FUNCTION_BLOCK FB_GetCPUTemp
VAR_INPUT
	rInterval			: REAL := 10.0;		// [sec]
END_VAR
VAR_OUTPUT
	rCPUTemp			: REAL;				// [deg]
	bError				: BOOL;				// error flag (indicator: error occured)
	nErrID				: UDINT;			// last error ID 
END_VAR
VAR
	// internal use
	sAmsNetId			: STRING := '';		// ADS Net ID (local = '')    
	iState				: INT;
	uData				: UINT;
	stMDP_Addr			: Tc2_MDP.ST_MDP_Addr;
	// FB instances
	fbReadMDPElement	: Tc2_MDP.FB_MDP_ReadElement;  
	tonInterval			: Tc2_Standard.TON;
END_VAR


// Interval timer
tonInterval(IN := NOT tonInterval.Q, PT := REAL_TO_TIME(rInterval * 1000.0));

CASE iState OF
	0: // Initiate program parameters (if required)
		fbReadMDPElement(bExecute := FALSE);
		IF (tonInterval.Q) THEN
			iState := 10;
		END_IF

	10:	// Trigger FB: request CPU data
		stMDP_Addr.nArea := INT_TO_BYTE(Tc2_MDP.eMDP_Area_ConfigArea);
		stMDP_Addr.nTableId := 1;
		stMDP_Addr.nSubIdx := 3;
		fbReadMDPElement(	bExecute := TRUE,
							eModuleType := Tc2_MDP.eMDP_ModT_CPU,
							stMDP_Addr := stMDP_Addr,
							iModIdx := 0,
							pDstBuf := ADR(uData),
							cbDstBufLen := SIZEOF(uData),
							sAmsNetId := sAmsNetId	);
		iState := 20;

	20:	// Process FB: Request CPU temp
		fbReadMDPElement(bExecute := FALSE); 
		IF (NOT fbReadMDPElement.bBusy) THEN
			IF (fbReadMDPElement.bError) THEN
				bError := TRUE;
				nErrID := fbReadMDPElement.nErrID; 
				iState := 0;
			ELSE
				bError := FALSE;
				rCPUTemp := UINT_TO_REAL(uData);
				iState := 30;
			END_IF                                               
		END_IF
    
     30: // Done 
		iState := 0;

	ELSE
		iState := 0; 

END_CASE

END_FUNCTION_BLOCK

(* stored: Version 1.1.0.1, ProductVersion 3.1.4024.2
   POU FB_GetCPUTemp: Id {07df4ad7-a000-41e9-baec-9c9601f89979}, SpecialFunc None *)
